INTERFACE IAbortableProcess EXTENDS IProcess

{attribute 'monitoring' := 'call'}
{attribute 'OPC.UA.DA.Property' := '1'}
{attribute 'OPC.UA.DA.Access' := '1'}
PROPERTY Aborted : BOOL
GET
END_GET
END_PROPERTY

{attribute 'monitoring' := 'call'}
{attribute 'OPC.UA.DA.Property' := '1'}
{attribute 'OPC.UA.DA.Access' := '1'}
PROPERTY AbortReason : REFERENCE TO ERROR_MESSAGE
GET
END_GET
END_PROPERTY

{attribute 'monitoring' := 'call'}
{attribute 'OPC.UA.DA.Property' := '1'}
{attribute 'OPC.UA.DA.Access' := '1'}
PROPERTY Busy : BOOL
GET
END_GET
END_PROPERTY

METHOD RequestAbort
VAR_INPUT 
	reason : ERROR_MESSAGE;
END_VAR
END_METHOD

END_INTERFACE

(* stored: Version 1.1.0.1
   Itf IAbortableProcess: Id {673acb26-d0c2-4ba2-81ae-6136dc542627}
   Property Aborted: Id {1b200195-722a-477c-8d67-52804e0bbba2}
   Get Get: Id {2472e367-f7fc-46ae-95ec-96cab3351e7b}
   Property AbortReason: Id {14a1cb54-5441-457c-bea8-c28e366481bc}
   Get Get: Id {de5e06a5-9fa3-434b-ba32-89384ee72df0}
   Property Busy: Id {2b26ebe6-1f26-4fe6-a5c9-8d70032d8fd6}
   Get Get: Id {a002431a-9e70-4409-840e-bad73d5c7158}
   Method RequestAbort: Id {8c3c78ee-be09-40e9-9b9f-fa08ff8e2858} *)
